FUNCTION GetMajor : UINT
VAR_INPUT
END_VAR
VAR
END_VAR

GetMajor := Version.Major;

END_FUNCTION

(* stored: Version 1.1.0.1, ProductVersion 3.1.4024.0
   POU GetMajor: Id {d7a5f597-3390-4262-a014-c48366ed1eef}, SpecialFunc None *)
